// TIA Portal V19 export
TYPE "C501_STU_IF_BBP_TYPIC"
   STRUCT
      CMD { ExternalAccessible := 'False'; ExternalVisible := 'False'; ExternalWritable := 'False'} : Bool;   // Aansturing pomp (TRUE = Aan / FALSE = Uit)
      LCK_AAN { ExternalAccessible := 'False'; ExternalVisible := 'False'; ExternalWritable := 'False'} : Bool;   // TRUE = Vergrendelen pomp (ook in manueel en hand)
      CMD_RES { ExternalAccessible := 'False'; ExternalVisible := 'False'; ExternalWritable := 'False'} : Bool;   // Reset van de latched storingen
   END_STRUCT;
END_TYPE
